FUNCTION_BLOCK Switch
VAR_INPUT
END_VAR
VAR_OUTPUT
END_VAR
VAR
END_VAR

METHOD PUBLIC IsPressed : BOOL
VAR_INPUT
END_VAR
END_METHOD

END_FUNCTION_BLOCK

(* stored: Version 1.1.0.1
   POU Switch: Id {a0cb1bcd-01f9-4361-a31e-d79f49bbe391}, SpecialFunc None
   Method IsPressed: Id {782b38c9-18b2-4323-a331-ba68dd02b06f} *)
